{attribute addProperty BoxType "EJ3214-0000-0016"}
{attribute addProperty Id "StatusAT %I*Status_C3A5DD7C1621ValueAT %I*INT16217"}
{attribute addProperty CRC "397281499"}
{attribute addProperty SizeInBites "32"}
{attribute addProperty SizeInBytes "4"}
TYPE RTD_Inputs_Channel_17AE08DB :
STRUCT
	{attribute addProperty Name "Status"}
	Status AT %I* : Status_C3A5DD7C;
	{attribute addProperty Name "Value"}
	Value AT %I* : INT;
END_STRUCT
END_TYPE

(* stored: Version 1.2.0.0, ProductVersion 3.1.4024.9
   DUT RTD_Inputs_Channel_17AE08DB: Id {922cf650-b66a-4770-9982-ce4e5acaaa51} *)
